(* PLC project Unnamed, Unknown Unnamed 1 *)
(* stored: creationDateTime 2025-04-10T10:18:14, modificationDateTime 2025-04-10T10:33:27 *)

PROGRAM program0
  VAR
    Fault : BOOL;
    Lamp : BOOL;
    ToggleTime : TIME := T#5s;
    TON0 : TON;
    TOF0 : TOF;
  END_VAR

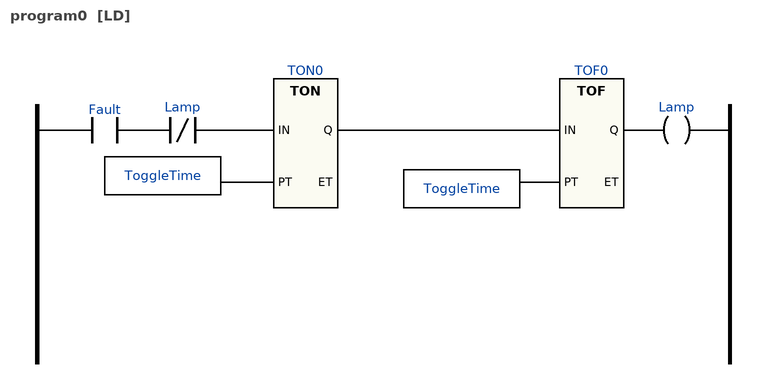
(* LD diagram, written out as Structured Text *)
TON0(IN := Fault AND NOT Lamp, PT := ToggleTime);
TOF0(IN := TON0.Q, PT := ToggleTime);
Lamp := TOF0.Q;
END_PROGRAM

CONFIGURATION Config0
  RESOURCE Res0 ON PLC
    TASK task0(INTERVAL := T#20ms, PRIORITY := 0);
    PROGRAM instance0 WITH task0 : program0;
  END_RESOURCE
END_CONFIGURATION
